INTERFACE I_Observer

METHOD M_Attach : BOOL
VAR_INPUT
	Object: 	I_Component;
END_VAR
END_METHOD

METHOD M_Detach : BOOL
VAR_INPUT
	Object: 	I_Component;
END_VAR
END_METHOD

METHOD M_Notify : BOOL
VAR_INPUT
	eRequest:		E_Request;
END_VAR
END_METHOD

END_INTERFACE

(* stored: Version 1.1.0.1
   Itf I_Observer: Id {af54216d-3f5e-4287-8176-18b478632bd5}
   Method M_Attach: Id {e1012f71-0b48-4ada-ba34-823492d9c2fe}
   Method M_Detach: Id {e09cef4f-639e-464f-affe-bde457fdaa63}
   Method M_Notify: Id {e795d50b-4d66-41e5-abd4-e88634350bb6} *)
